{attribute 'qualified_only'}
{attribute 'strict'}
TYPE E_Error :
(
	OK := 0,
    SomeError := 5,
    OtherError
) USINT;
END_TYPE

(* stored: Version 1.1.0.1, ProductVersion 3.1.4024.11
   DUT E_Error: Id {c568c63f-be9a-4c9b-92a0-4c4517e2c530} *)
